TYPE ST_DLK_Parameter :
STRUCT


	Temp_Warmwasser	       : REAL;
	Temp_Warmwasser_Max    : REAL;
	Temp_Warmwasser_Min    : REAL;


	AutoQuittierung			: BOOL;

END_STRUCT
END_TYPE

(* stored: Version 1.1.0.1, ProductVersion 3.1.4024.9
   DUT ST_DLK_Parameter: Id {4eb37ad5-8639-4611-98fd-9dc32185f0c9} *)
